FUNCTION WRITE_ANY_UINT : BOOL
VAR_INPUT
    ptr: POINTER TO UINT;
    val: UINT;
END_VAR

ptr^ := val;

END_FUNCTION

(* stored: Version 1.1.0.1, ProductVersion 3.1.4022.9
   POU WRITE_ANY_UINT: Id {4b5114b2-1dc0-4e59-81df-bbfea3eeaaa0}, SpecialFunc None *)
